FUNCTION_BLOCK "FB_CalculateDayOfYear"
{ S7_Optimized_Access := 'TRUE' }
   VAR_INPUT
      Year : INT;
      Month : INT;
      Day : INT;
   END_VAR

   VAR_OUTPUT
      DayOfYear : INT;
      error : BOOL;
      status : WORD;
   END_VAR

   VAR
      DaysInMonth : ARRAY[1..12] OF INT := [31, 28, 31, 30, 31, 30, 31, 31, 30, 31, 30, 31];
      i: INT;
   END_VAR

BEGIN
   // Initialize outputs
   #DayOfYear := 0;
   #error := FALSE;
   #status := 0;

   // Check for valid year
   IF (#Year < 1000) OR (#Year > 3000) THEN
      #error := TRUE;
      #status := 16#8001;
      RETURN;
   END_IF;

   // Check for valid month
   IF (#Month < 1) OR (#Month > 12) THEN
      #error := TRUE;
      #status := 16#8002;
      RETURN;
   END_IF;

   // Adjust February days for leap year
   IF (#Year MOD 4 = 0) AND (NOT (#Year MOD 100 = 0)) OR (#Year MOD 400 = 0) THEN
      #DaysInMonth[2] := 29;
   ELSE
      #DaysInMonth[2] := 28;
   END_IF;

   // Check for valid day
   IF (#Day < 1) OR (#Day > #DaysInMonth[Month]) THEN
      #error := TRUE;
      #status := 16#8003;
      RETURN;
   END_IF;

   // Calculate DayOfYear
   FOR #i := 1 TO #Month-1 DO
      #DayOfYear := #DayOfYear + #DaysInMonth[i];
   END_FOR;
   #DayOfYear := #DayOfYear + #Day;

END_FUNCTION_BLOCK
